PROGRAM MAIN
VAR
END_VAR

END_PROGRAM

(* stored: Version 1.1.0.1
   POU MAIN: Id {a2905053-aeab-4090-9af5-e3971c4ed8f3} *)
